// TwinCAT 3 PLC project LF_System_PLC
// ProgramVersion: 3.1.4026.21
// CompilerDefines: VISU_USEPROPERTYINFO
// libraries:
//   Tc2_Standard, * (Beckhoff Automation GmbH)
//   Tc2_System, * (Beckhoff Automation GmbH)
//   Tc3_IotBase, * (Beckhoff Automation GmbH)
//   VisuSymbols, 4.5.0.0 (System)
// project tree:
//   DUTs/ Betriebszustand.TcDUT
//   / GlobalTextList.TcGTLO (not stored), PlcTask.TcTTO (not stored), Visualization Manager.TcVMO (not stored)
//   POUs/Extruder/ FB_System_FlaschenFullstand.TcPOU (not stored), FB_System_Fullstand.TcPOU (not stored)
//   POUs/Förderband/ FB_System_CNV.TcPOU (not stored)
//   POUs/ MAIN.TcPOU (not stored)
//   POUs/Manipulator/ FB_System_LinAxis.TcPOU
//   POUs/Vereinzelung/ FB_SpeicherRohr.TcPOU (not stored), FB_System_Vereinzelung.TcPOU (not stored)
//   VISUs/ Visualization.TcVIS
// (motion and I/O tree: see PLC project tempmodel)
// real-time tasks:
//   TASK PlcTask: cycle T#10ms, priority 21, ADS port 350
//   TASK PlcTask1: cycle T#10ms, priority 22, ADS port 351
//   TASK PlcTask2: cycle T#10ms, priority 20, ADS port 352
// variable links:
//   LF_System_PLC/LF_System_PLC Instance <-> NC-Task 1 SAF/Axes/BandAchse
//     PlcTask Inputs/MAIN.fIN_CnvPos <-> Outputs/ToPlc/ActPos
//   LF_System_PLC/LF_System_PLC Instance <-> NC-Task 1 SAF/Axes/Extruder1
//     PlcTask Inputs/MAIN.fIN_ExtPos1 <-> Outputs/ToPlc/ActPos
//   LF_System_PLC/LF_System_PLC Instance <-> NC-Task 1 SAF/Axes/Extruder2
//     PlcTask Inputs/MAIN.fIN_ExtPos2 <-> Outputs/ToPlc/ActPos
//   LF_System_PLC/LF_System_PLC Instance <-> NC-Task 1 SAF/Axes/Extruder3
//     PlcTask Inputs/MAIN.fIN_ExtPos3 <-> Outputs/ToPlc/ActPos
//   LF_System_PLC/LF_System_PLC Instance <-> NC-Task 1 SAF/Axes/X_Achse_Manipulator
//     PlcTask Inputs/MAIN.fIN_ManXPos <-> Outputs/ToPlc/ActPos
//   LF_System_PLC/LF_System_PLC Instance <-> PLC/PLC Instance
//     PlcTask Inputs/MAIN.bIN_Gripper <-> PlcTask Outputs/IFC_HW.bGripperClosed
//     PlcTask Inputs/MAIN.bIN_Stopper1 <-> PlcTask Outputs/IFC_HW.bBandHub1
//     PlcTask Inputs/MAIN.bIN_Stopper2 <-> PlcTask Outputs/IFC_HW.bBandHub2
//     PlcTask Inputs/MAIN.bIN_Stopper3 <-> PlcTask Outputs/IFC_HW.bBandHub3
//     PlcTask Inputs/MAIN.bIn_LedGreen <-> PlcTask Outputs/IFC_HW.bAmpelGrun
//     PlcTask Inputs/MAIN.bIn_LedRot <-> PlcTask Outputs/IFC_HW.bAmpelRot
//     PlcTask Inputs/MAIN.bIn_LedYellow <-> PlcTask Outputs/IFC_HW.bAmpelGelb
//     PlcTask Inputs/MAIN.bIn_Schleuse1_L1 <-> PlcTask Outputs/IFC_HW.bR1AKT1
//     PlcTask Inputs/MAIN.bIn_Schleuse1_L2 <-> PlcTask Outputs/IFC_HW.bR2AKT1
//     PlcTask Inputs/MAIN.bIn_Schleuse2_L1 <-> PlcTask Outputs/IFC_HW.bR1AKT2
//     PlcTask Inputs/MAIN.bIn_Schleuse2_L2 <-> PlcTask Outputs/IFC_HW.bR2AKT2
//     PlcTask Outputs/MAIN.bEnable <-> PlcTask Inputs/IFC_HW.bEnable
//     PlcTask Outputs/MAIN.bExecute <-> PlcTask Inputs/IFC_HW.bExecute
//     PlcTask Outputs/MAIN.bOUT_CnvNS{1..4} <-> PlcTask Inputs/IFC_HW.bBandSens{1..4}  (4 links)
//     PlcTask Outputs/MAIN.bOUT_SensMaxX <-> PlcTask Inputs/IFC_HW.bManEndXmax
//     PlcTask Outputs/MAIN.bOUT_SensMinX <-> PlcTask Inputs/IFC_HW.bManEndXmin
//     PlcTask Outputs/MAIN.bOut_VereinzelungNS1 <-> PlcTask Inputs/IFC_HW.bEinzelSens1
//     PlcTask Outputs/MAIN.bOut_VereinzelungNS2 <-> PlcTask Inputs/IFC_HW.bEinzelSens2
//     PlcTask Outputs/MAIN.bOut_VereinzelungNS3 <-> PlcTask Inputs/IFC_HW.bEinzelSens3
//     PlcTask Outputs/MAIN.iOut_USS1 <-> PlcTask Inputs/IFC_HW.iFillSens1
//     PlcTask Outputs/MAIN.iOut_USS2 <-> PlcTask Inputs/IFC_HW.iFillSens2
//     PlcTask Outputs/MAIN.iOut_USS3 <-> PlcTask Inputs/IFC_HW.iFillSens3

// ---- DUTs/Betriebszustand.TcDUT
{attribute 'qualified_only'}
{attribute 'strict'}
{attribute 'to_string'}
TYPE Betriebszustand :
(
	Aus,
	Produktion,
	Fehler,
	Warnung,
	Init,
	Bereit,
	Fertig
);
END_TYPE

// ---- POUs/Manipulator/FB_System_LinAxis.TcPOU
FUNCTION_BLOCK FB_System_LinAxis
VAR_INPUT
	fPos : LREAL;
	bGripperOpen : BOOL;
	PosSensMin : INT;
	PosSensMax : INT;
END_VAR
VAR_OUTPUT
	bSensMin : BOOL;
	bSensMax : BOOL;
END_VAR
VAR
	iBottlePosX : INT;
	iAxPos: INT;
	fAxPosOff : LREAL;
	
	nState : INT := 0;
	rTrig : F_Trig;
END_VAR

IF iAxPos <= -189 THEN
	bSensMin := FALSE;
	bSensMax := TRUE;
ELSIF iAxPos >= 241 THEN
	bSensMin := TRUE;
	bSensMax := FALSE;
ELSE
	bSensMin := TRUE;
	bSensMax := TRUE;
END_IF


// State Machine Implementieren...
CASE nState OF
// Offset differenz bei Homing
0:
IF fPos > 9999999900 THEN
	fAxPosOff := 9999999999.9999;
ELSIF fPos < -9999999900 THEN
	fAxPosOff := -9999999999.9999;
ELSIF fPos < 9990000000 AND fPos > -9999999000 THEN
	fAxPosOff := 0;
END_IF

rTrig(CLK:= NOT bSensMin, Q=>);
IF rTrig.Q  THEN
	nState := 1;
END_IF

1:

IF fPos > -999999 AND fpos < 999999 THEN
	fAxPosOff := 269; // falscher Offset!!!!
END_IF

END_CASE


IF fPos-fAxPosOff > 9999999990 OR fPos-fAxPosOff < -9999999990 THEN
	iAxPos := 0;
ELSE
	iAxPos := TO_INT((fPos-fAxPosOff) * 0.7);
END_IF

IF NOT bGripperOpen THEN
	iBottlePosX := iAxPos;
END_IF

END_FUNCTION_BLOCK

// ---- VISUs/Visualization.TcVIS
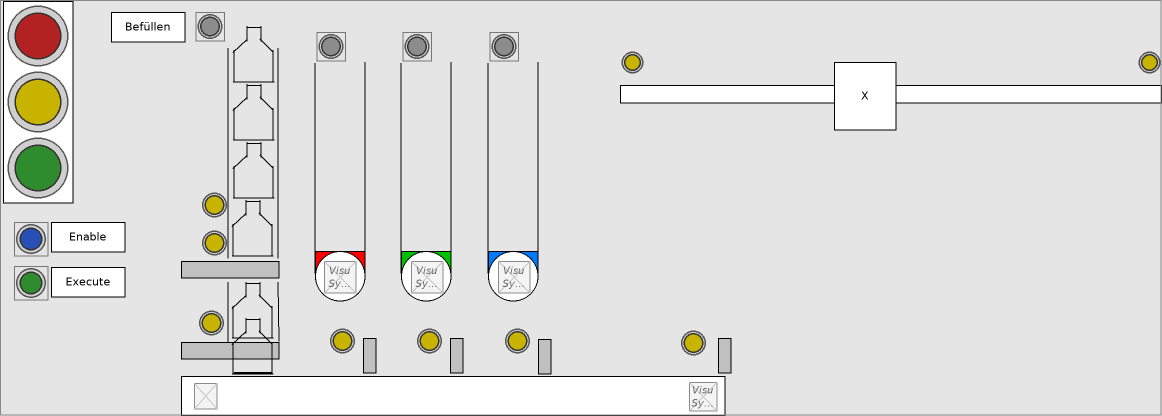
VISUALIZATION Visualization  // 1162x416
    Rectangle (315,251 50x24)
        p2773130477: - MAIN.fbExt1.iFillLevel
    Lamp1 (200,190 29x30), variable: MAIN.bOut_VereinzelungNS1, style: Lamp-Lamp1-Yellow
    Lamp1 (200,228 29x30), variable: MAIN.bOut_VereinzelungNS2, style: Lamp-Lamp1-Yellow
    Lamp1 (197,308 29x30), variable: MAIN.bOut_VereinzelungNS3, style: Lamp-Lamp1-Yellow
    Group (3,1 70x202)
        Rectangle (0,0 70x202)
        Lamp1 (0,0 70x70), variable: MAIN.bIn_LedRot, style: Lamp-Lamp1-Red
        Lamp1 (0,66 70x70), variable: MAIN.bIn_LedYellow, style: Lamp-Lamp1-Yellow
        Lamp1 (0,132 70x70), variable: MAIN.bIn_LedGreen, style: Lamp-Lamp1-Green
    Line (228,258) (228,48)
    Line (278,258) (278,48)
    Line (279,341) (278,282)
    Line (228,342) (228,282)
    Rectangle (181,261 98x17)
        p3528305787: MAIN.fbVereinzelung.S1pos
        p874137650: MAIN.fbVereinzelung.S1pos
    Rectangle (181,342 98x17)
        p3528305787: MAIN.fbVereinzelung.S2pos
        p874137650: MAIN.fbVereinzelung.S2pos
    PushSwitch (12,222 38x34), variable: MAIN.bEnable, behaviour: TOGGLE, style: Switch-PushSwitch-Blue
    PushSwitch (12,266 38x34), variable: MAIN.bExecute, behaviour: TAP, style: Switch-PushSwitch-Green
    Rectangle (51,222 74x30), "Enable"
    Rectangle (51,267 74x30), "Execute"
    Group (232,200 41x57), invisible if: not MAIN.fbVereinzelung.fbSpeicherRohr.aSpeicher[0]
        Line (1,56) (1,24)
        Line (40,55) (40,24)
        Line (41,56) (0,56)
        Line (0,26) (14,13)
        Line (40,26) (27,13)
        Line (14,15) (14,0)
        Line (28,15) (28,0)
        Line (14,1) (28,1)
    Group (233,142 41x57), invisible if: Not MAIN.fbVereinzelung.fbSpeicherRohr.aSpeicher[1]
        Line (1,56) (1,24)
        Line (40,55) (40,24)
        Line (41,56) (0,56)
        Line (0,26) (14,13)
        Line (40,26) (27,13)
        Line (14,15) (14,0)
        Line (28,15) (28,0)
        Line (14,1) (28,1)
    Group (232,282 41x57), invisible if: not MAIN.bOut_VereinzelungNS3
        Line (1,56) (1,24)
        Line (40,55) (40,24)
        Line (41,56) (0,56)
        Line (0,26) (14,13)
        Line (40,26) (27,13)
        Line (14,15) (14,0)
        Line (28,15) (28,0)
        Line (14,1) (28,1)
    Group (233,84 41x57), invisible if: Not MAIN.fbVereinzelung.fbSpeicherRohr.aSpeicher[2]
        Line (1,56) (1,24)
        Line (40,55) (40,24)
        Line (41,56) (0,56)
        Line (0,26) (14,13)
        Line (40,26) (27,13)
        Line (14,15) (14,0)
        Line (28,15) (28,0)
        Line (14,1) (28,1)
    Group (233,26 41x57), invisible if: Not MAIN.fbVereinzelung.fbSpeicherRohr.aSpeicher[3]
        Line (1,56) (1,24)
        Line (40,55) (40,24)
        Line (41,56) (0,56)
        Line (0,26) (14,13)
        Line (40,26) (27,13)
        Line (14,15) (14,0)
        Line (28,15) (28,0)
        Line (14,1) (28,1)
    PushSwitch (194,12 32x29), variable: MAIN.fbVereinzelung.bBefullen, behaviour: TAP, style: Switch-PushSwitch-Gray
    RoundedRectangle (181,376 544x40)
    Lamp1 (328,326 29x30), variable: MAIN.bOUT_CnvNS1, style: Lamp-Lamp1-Yellow
    Lamp1 (503,326 29x30), variable: MAIN.bOUT_CnvNS3, style: Lamp-Lamp1-Yellow
    Lamp1 (415,326 29x30), variable: MAIN.bOUT_CnvNS2, style: Lamp-Lamp1-Yellow
    Lamp1 (679,328 29x30), variable: MAIN.bOUT_CnvNS4, style: Lamp-Lamp1-Yellow
    Group (232,318 41x57), invisible if: not MAIN.fbCNV.bBottleOnCNV
        p3560616238: MAIN.fbCNV.iBottlePos
        Line (1,56) (1,24)
        Line (40,55) (40,24)
        Line (41,56) (0,56)
        Line (0,26) (14,13)
        Line (40,26) (27,13)
        Line (14,15) (14,0)
        Line (28,15) (28,0)
        Line (14,1) (28,1)
    Rectangle (363,338 13x35), invisible if: MAIN.bIN_Stopper1
    Rectangle (450,338 13x35), invisible if: MAIN.bIN_Stopper2
    Rectangle (538,339 13x35), invisible if: MAIN.bIN_Stopper3
    Rectangle (718,338 13x35)
    Image (194,383 23x26), invisible if: not MAIN.fbCNV.bCNVisMoving, image: VisuSymbols.Symbols.ArrowHalfRightUp
    Image (689,382 28x29), invisible if: not MAIN.fbCNV.bCNVisMoving, image: VisuSymbols.Symbols.ArrowHalfRightDown
    Rectangle (111,12 74x30), "Befüllen"
    Ellipse (315,251 50x50)
    Line (315,273) (315,63)
    Line (365,272) (365,62)
    Rectangle (401,251 50x24)
        p2773130477: - MAIN.fbExt2.iFillLevel
    Ellipse (401,251 50x50)
    Line (401,273) (401,63)
    Line (451,272) (451,62)
    Rectangle (488,251 50x24)
        p2773130477: - MAIN.fbExt3.iFillLevel
    Ellipse (488,251 50x50)
    Line (488,273) (488,63)
    Line (538,272) (538,62)
    PushSwitch (315,32 32x29), variable: MAIN.bRefill1, behaviour: TAP, style: Switch-PushSwitch-Gray
    PushSwitch (401,32 32x29), variable: MAIN.bRefill2, behaviour: TAP, style: Switch-PushSwitch-Gray
    PushSwitch (488,32 32x29), variable: MAIN.bRefill3, behaviour: TAP, style: Switch-PushSwitch-Gray
    Image (324,261 32x32), invisible if: MAIN.fbExt1.NotMoving, image: VisuSymbols.Symbols.ArrowCircle2RightRightLeft
    Image (411,261 32x32), invisible if: MAIN.fbExt2.NotMoving, image: VisuSymbols.Symbols.ArrowCircle2RightRightLeft
    Image (498,261 32x32), invisible if: MAIN.fbExt3.NotMoving, image: VisuSymbols.Symbols.ArrowCircle2RightRightLeft
    Rectangle (234,372 38x1), invisible if: not MAIN.fbCNV.bBottleOnCNV
        p2773130477: - MAIN.fbBottleLevel.iFillLevel3 - MAIN.fbBottleLevel.iFillLevel1 - MAIN.fbBottleLevel.iFillLevel2
        p3560616238: MAIN.fbCNV.iBottlePos
        p1126004900: - MAIN.fbBottleLevel.iFillLevel1 - MAIN.fbBottleLevel.iFillLevel2
    Rectangle (234,372 38x1), invisible if: not MAIN.fbCNV.bBottleOnCNV
        p2773130477: - MAIN.fbBottleLevel.iFillLevel2 - MAIN.fbBottleLevel.iFillLevel1
        p3560616238: MAIN.fbCNV.iBottlePos
        p1126004900: - MAIN.fbBottleLevel.iFillLevel1
    Rectangle (234,372 38x1), invisible if: not MAIN.fbCNV.bBottleOnCNV
        p2773130477: - MAIN.fbBottleLevel.iFillLevel1
        p3560616238: MAIN.fbCNV.iBottlePos
    Rectangle (620,85 542x18)
    Rectangle (834,62 62x68), "X"
        p3560616238: MAIN.fbManAxX.iAxPos
    Lamp1 (620,50 25x25), variable: MAIN.bOUT_SensMinX, style: Lamp-Lamp1-Yellow
    Lamp1 (1137,50 25x25), variable: MAIN.bOUT_SensMaxX, style: Lamp-Lamp1-Yellow
END_VISUALIZATION
